// TwinCAT 3 PLC project Controller
// ProgramVersion: 3.1.4026.15
// libraries:
//   Tc2_Math, * (Beckhoff Automation GmbH)
//   Tc2_MC2, * (Beckhoff Automation GmbH)
//   Tc2_MC2_Camming, * (Beckhoff Automation GmbH)
//   Tc2_Standard, * (Beckhoff Automation GmbH)
//   Tc2_System, * (Beckhoff Automation GmbH)
//   Tc2_Utilities, * (Beckhoff Automation GmbH)
//   Tc3_Module, * (Beckhoff Automation GmbH)
// project tree:
//   DUTs/ ST_RECIPE_VARIABLES.TcDUT, ST_WORKER_VARIABLES.TcDUT
//   GVLs/ GVL.TcGVL
//   / PlcTask.TcTTO
//   POUs/ FB_CamProfiles.TcPOU, FB_MasterCamControl.TcPOU, MAIN.TcPOU
// real-time tasks:
//   TASK PlcTask: cycle T#10ms, priority 20, ADS port 350
// motion (NC):
//   TASK NC-Task 1 SAF: cycle T#2ms, priority 4, ADS port 501
//   TASK NC-Task 1 SVB: cycle T#10ms, priority 8, ADS port 511
//   AXIS Master (id 1)
//     Velo: Maximum=10000
//     OtherSettings: AllowMotionCmdToSlave=true
//     encoder EncType=1
//     drive DrvType=5
//       Analog: TorqueSetpointScale=10, ScaleFactorActTorque=0.1
//       TimeComp: TaskDelayCycles=1
//     controller CtrType=1
//       CtrPara: PriorControlFactor=1
//         Observer: BandWidth=20
//   AXIS Slave_1 (id 2)
//     OtherSettings: AllowMotionCmdToSlave=true
//     encoder EncType=1
//     drive DrvType=5
//       Analog: TorqueSetpointScale=10, ScaleFactorActTorque=0.1
//       TimeComp: TaskDelayCycles=1
//     controller CtrType=1
//       CtrPara: PriorControlFactor=1
//         Observer: BandWidth=20
//   AXIS Slave_2 (id 3)
//     OtherSettings: AllowMotionCmdToSlave=true
//     encoder EncType=1
//     drive DrvType=5
//       Analog: TorqueSetpointScale=10, ScaleFactorActTorque=0.1
//       TimeComp: TaskDelayCycles=1
//     controller CtrType=1
//       CtrPara: PriorControlFactor=1
//         Observer: BandWidth=20
//   AXIS Slave_3 (id 4)
//     OtherSettings: AllowMotionCmdToSlave=true
//     encoder EncType=1
//     drive DrvType=5
//       Analog: TorqueSetpointScale=10, ScaleFactorActTorque=0.1
//       TimeComp: TaskDelayCycles=1
//     controller CtrType=1
//       CtrPara: PriorControlFactor=1
//         Observer: BandWidth=20
//   AXIS Slave_4 (id 5)
//     OtherSettings: AllowMotionCmdToSlave=true
//     encoder EncType=1
//     drive DrvType=5
//       Analog: TorqueSetpointScale=10, ScaleFactorActTorque=0.1
//       TimeComp: TaskDelayCycles=1
//     controller CtrType=1
//       CtrPara: PriorControlFactor=1
//         Observer: BandWidth=20
// variable links:
//   Controller/Controller Instance <-> NC-Task 1 SAF/Axes/Master
//     PlcTask Inputs/GVL.Master.NcToPlc <-> Outputs/ToPlc
//     PlcTask Outputs/GVL.Master.PlcToNc <-> Inputs/FromPlc
//   Controller/Controller Instance <-> NC-Task 1 SAF/Axes/Slave_1
//     PlcTask Inputs/GVL.Slave_1.NcToPlc <-> Outputs/ToPlc
//     PlcTask Outputs/GVL.Slave_1.PlcToNc <-> Inputs/FromPlc
//   Controller/Controller Instance <-> NC-Task 1 SAF/Axes/Slave_2
//     PlcTask Inputs/GVL.Slave_2.NcToPlc <-> Outputs/ToPlc
//     PlcTask Outputs/GVL.Slave_2.PlcToNc <-> Inputs/FromPlc
//   Controller/Controller Instance <-> NC-Task 1 SAF/Axes/Slave_3
//     PlcTask Inputs/GVL.Slave_3.NcToPlc <-> Outputs/ToPlc
//     PlcTask Outputs/GVL.Slave_3.PlcToNc <-> Inputs/FromPlc
//   Controller/Controller Instance <-> NC-Task 1 SAF/Axes/Slave_4
//     PlcTask Inputs/GVL.Slave_4.NcToPlc <-> Outputs/ToPlc
//     PlcTask Outputs/GVL.Slave_4.PlcToNc <-> Inputs/FromPlc

CONFIGURATION Controller
    RESOURCE PLC ON TwinCAT3
        TASK PlcTask(INTERVAL := T#10ms, PRIORITY := 20);
        PROGRAM MAIN WITH PlcTask : MAIN;
    END_RESOURCE
END_CONFIGURATION

// ---- DUTs/ST_RECIPE_VARIABLES.TcDUT
TYPE ST_RECIPE_VARIABLES :
STRUCT
	sRecipeName			: STRING;
	MotionPoints_CAM_1	: ARRAY [0..360, 0..1] OF REAL;
	MotionPoints_CAM_2	: ARRAY [0..360, 0..1] OF REAL;
	MotionPoints_CAM_3	: ARRAY [0..360, 0..1] OF REAL;
	MotionPoints_CAM_4	: ARRAY [0..360, 0..1] OF REAL;
	// And other Recipe Variables
	bCheckBool			: BOOL;
	nTestInt			: INT;
	rTestReal			: REAL;
	lrTestLReal			: LREAL;
	udnAnotherInt		: UDINT;
END_STRUCT
END_TYPE

// ---- DUTs/ST_WORKER_VARIABLES.TcDUT
TYPE ST_WORKER_VARIABLES :
STRUCT
	sMachineName		: STRING := 'Worker_1';
	sProgramVersion		: STRING := '1.0';
	stRecipeVariables	: ST_RECIPE_VARIABLES;
	
	eStatus				: (IDLE,
							ASSIGNED,
							RUNNING,
							MAINTAINANCE_REQ);
	
	bGetRecipeAndCams	: BOOL;
	bCamsReady			: BOOL;
	sAssignedRecipe		: STRING;
	udnNumberOfJobsDone	: UDINT;
	udnDaysSinceServiced: UDINT;
END_STRUCT
END_TYPE

// ---- GVLs/GVL.TcGVL
{attribute 'qualified_only'}
VAR_GLOBAL
	Master		: AXIS_REF;		// Master will be a virtual axis
	rMasterVel	: REAL;
	
	// The 4 slaves will be the 4 Beckhoff motors
	Slave_1		: AXIS_REF;
	Slave_2		: AXIS_REF;
	Slave_3		: AXIS_REF;
	Slave_4		: AXIS_REF;
END_VAR

// ---- POUs/MAIN.TcPOU
PROGRAM MAIN
VAR
	stWorker_1		: ST_WORKER_VARIABLES;
	stRecipe		: ST_RECIPE_VARIABLES;
	
	// Slave positions for the cam table
	// Array [1..4] are slaves 1 - 4, each of the slave is a 2d array **REQUIRED by cam table ref**
	// Array [0..359] are master-slave position pair
	ALL_CAM			: ARRAY [1..4] OF ARRAY [0..359] OF ARRAY [0..1] OF LREAL;		
	ALL_CAM_REF		: ARRAY [1..4] OF MC_CAM_REF;		// Cam table reference
	
	nState			: INT;
	bStart			: BOOL;
	
	fbMasterCam		: FB_MasterCamControl;
	fbCamProfiles	: FB_CamProfiles;
	mcHome			: MC_Home;
	bMasterRun		: BOOL;
	bHalt			: BOOL;
	bReset			: BOOL;
	bReadDone		: BOOL;
	bCreateDone		: BOOL;
	
	bCamIn			: BOOL;
	nUpdate			: INT;
END_VAR

fbMasterCam();

CASE nState OF
	0:	// IDLE
		IF bStart THEN
			nState		:= 5;
		END_IF
	5:	// Initialize and enable the power on Master and Slaves Axes
		fbMasterCam.mInitialize(TRUE);
		IF fbMasterCam.pInitialized THEN
			fbMasterCam.mInitialize(FALSE);
			nState		:= 10;
		END_IF
	(**************** These will not be implemented in the real project ***********)
	(**************** recipe management will replace the csv file *****************)
	10:	// Read CAM profiles from CSV files and store in CAM arrays
		fbCamProfiles.mReadAndStoreSlavePositions(TRUE, ALL_CAM);
		IF fbCamProfiles.pReadDone THEN
			fbCamProfiles.mReadAndStoreSlavePositions(FALSE, ALL_CAM);
			nState		:= 15;
		END_IF
	15:	// Create Twincat digital CAM tables from CAM profile arrays
		fbCamProfiles.mCreateCamProfiles(TRUE, ALL_CAM, ALL_CAM_REF);
		IF fbCamProfiles.pCreateDone THEN
			fbCamProfiles.mCreateCamProfiles(FALSE, ALL_CAM, ALL_CAM_REF);
			GVL.rMasterVel:= 0.5;			// Start Master at minimum speed
			bMasterRun	:= TRUE;			// to couple CAM profiles
			fbMasterCam.pRunCams:= TRUE;	// Start Slaves
			nState		:= 20;
		END_IF
	(**************      ~30s to complete the csv reading     *********************)
	(******************************************************************************)
	20:	// Assign CAM tables to their respective Slave Axes
		fbMasterCam.mMultiCamIn(TRUE);
		IF fbMasterCam.pCamInDone THEN
			fbMasterCam.mMultiCamIn(TRUE);
			nState		:= 25;
		END_IF
	25:	// Speed up Master after all CAMs done coupling 
		IF NOT bMasterRun THEN
			GVL.rMasterVel	:= 180;
			bMasterRun		:= TRUE;
			nState			:= 26;
		END_IF
		
	(********************* Not used *******************)
	30:	// Stop all axes
		fbMasterCam.mHalt(bHalt);
	35: // Reset all axes
		fbMasterCam.mReset(bReset);
END_CASE
fbMasterCam.mRun(bMasterRun);

METHOD mLoadCSVToCAMs : BOOL
//VAR_INPUT
//	Execute		: BOOL;
//END_VAR
//VAR_IN_OUT
//	Slave_CAM	: ARRAY [0..360] OF ARRAY [0..1] OF LREAL;
//END_VAR
//CASE nState OF
//	0:
//		IF Execute THEN
//			sReadLine	:= '';
//			nStringIndex:= 0;
//			nState		:= 1;
//		END_IF
//	1:
//		fbFileOpen(
//			sNetId		:= '10.75.0.183.1.1',
//			sPathName	:= sFilePath,
//			nMode		:= FOPEN_MODEREAD,
//			ePath		:= PATH_GENERIC,
//			bExecute	:= TRUE,
//			tTimeout	:= DEFAULT_ADS_TIMEOUT);
//		nState			:= 2;
//	2:
//		fbFileOpen(	
//			bExecute 	:= FALSE,
//			hFile 		=> fileHandle);
//		IF NOT fbFileOpen.bBusy THEN
//			IF NOT fbFileOpen.bError THEN
//				nState	:= 5;
//			ELSE
//				nState	:= 255;
//			END_IF
//		END_IF
//	5:
//		fbFileGets(
//			sNetId		:= '10.75.0.183.1.1',
//			hFile		:= fileHandle,
//			bExecute	:= TRUE,
//			sLine		=> sReadLine);
//		IF NOT fbFileGets.bBusy AND NOT fbFileGets.bError THEN
//			fbFileGets(bExecute:=FALSE);
//			IF NOT fbFileGets.bEOF THEN
//				nState	:= 10;
//			ELSE
//				nStringIndex:= 0;
//				nState	:= 15;
//			END_IF
//		ELSIF fbFileGets.bError THEN
//				nState	:= 255;
//		END_IF
//	10:
//		arrString[nStringIndex]:= sReadLine;
//		nStringIndex	:= nStringIndex + 1;
//		nState			:= 5;
//	15:
//		FOR nStringIndex := 0 TO 360 DO
//			rAbsPosition:= STRING_TO_REAL(arrString[nStringIndex]);
//			arrTemp[0]	:= nStringIndex;
//			arrTemp[1]	:= rAbsPosition;
//			Slave_CAM[nStringIndex]:= arrTemp;
//		END_FOR
//		nState			:= 60;
		
//	60:
//		fbFileClose(
//			sNetId		:= '10.75.0.183.1.1',
//			hFile		:= fileHandle,
//			bExecute	:= TRUE);
//		nState			:= 61;
//	61:
//		fbFileClose(bExecute:=FALSE);
//		IF NOT fbFileClose.bBusy THEN
//			IF NOT fbFileClose.bError THEN
//				nState	:= 62;
//			ELSE
//				nState	:= 255;
//			END_IF
//		END_IF
//	62:
//		sTemp			:= '';
//		sFilePath		:= 'C:\';
//		bExecute		:= FALSE;
//		nState			:= 0;
//END_CASE
END_METHOD

END_PROGRAM

// ---- POUs/FB_MasterCamControl.TcPOU
FUNCTION_BLOCK FB_MasterCamControl
VAR_INPUT
END_VAR
VAR_OUTPUT
END_VAR
VAR
//	fbMaster		: CAM_AXIS_BASE;
//	fbSlave_1		: CAM_AXIS_BASE;
//	fbSlave_2		: CAM_AXIS_BASE;
//	fbSlave_3		: CAM_AXIS_BASE;
//	fbSlave_4		: CAM_AXIS_BASE;
	mcHome			: MC_Home;
	bRunCams		: BOOL;
	
	bInitialized	: BOOL;
	bCamInDone		: BOOL;
END_VAR

//fbMaster.mRunCam(bRunCams);
//fbSlave_1.mRunCam(bRunCams);
//fbSlave_2.mRunCam(bRunCams);
//fbSlave_3.mRunCam(bRunCams);
//fbSlave_4.mRunCam(bRunCams);

// Reset Virtual Master Cam to 0 after 1 complete revolution
IF GVL.Master.NcToPlc.ModuloSetTurns = 1 AND NOT mcHome.Done THEN
	mcHome(
		Axis		:= GVL.Master,
		Execute		:= TRUE,
		Position	:= 0,
		HomingMode	:= MC_Direct);
ELSIF mcHome.Done THEN
	mcHome(Axis := GVL.Master, Execute := FALSE);
END_IF

METHOD mCamOut : BOOL
VAR_INPUT
	Execute		: BOOL;
END_VAR

VAR_INST
	CamOut		: MC_CamOut;
	
	nState		: INT;
	rtStart		: R_TRIG;
END_VAR
CASE nState OF
	0:
		rtStart(CLK := Execute);
		IF rtStart.Q THEN
			mCamOut		:= FALSE;
			nState		:= 5;
		END_IF
	5:
		CamOut(Slave := GVL.Slave_1, Execute := TRUE);
		IF CamOut.Done THEN
			CamOut(Slave := GVL.Slave_1, Execute := FALSE);
			nState		:= 15;
		END_IF
	15:
		CamOut(Slave := GVL.Slave_2, Execute := TRUE);
		IF CamOut.Done THEN
			CamOut(Slave := GVL.Slave_2, Execute := FALSE);
			nState		:= 20;
		END_IF
	20:
		CamOut(Slave := GVL.Slave_3, Execute := TRUE);
		IF CamOut.Done THEN
			CamOut(Slave := GVL.Slave_3, Execute := FALSE);
			nState		:= 25;
		END_IF
	25:
		CamOut(Slave := GVL.Slave_4, Execute := TRUE);
		IF CamOut.Done THEN
			CamOut(Slave := GVL.Slave_4, Execute := FALSE);
			nState		:= 30;
		END_IF
	30:
		mCamOut			:= TRUE;
		nState			:= 0;
END_CASE
END_METHOD

METHOD mHalt : BOOL
VAR_IN_OUT
	Execute		: BOOL;
END_VAR
VAR_INST
	HaltMaster	: MC_Halt;
	HaltSlave_1	: MC_Halt;
	HaltSlave_2	: MC_Halt;
	HaltSlave_3	: MC_Halt;
	HaltSlave_4	: MC_Halt;
END_VAR
HaltMaster(Axis := GVL.Master, Execute := Execute);
HaltSlave_1(Axis := GVL.Slave_1, Execute := Execute);
HaltSlave_2(Axis := GVL.Slave_2, Execute := Execute);
HaltSlave_3(Axis := GVL.Slave_3, Execute := Execute);
HaltSlave_4(Axis := GVL.Slave_4, Execute := Execute);

IF HaltMaster.Done AND HaltSlave_1.Done AND HaltSlave_2.Done AND HaltSlave_3.Done AND HaltSlave_4.Done THEN
	Execute := FALSE;
END_IF
END_METHOD

(* Move all axes to 0 position *)
METHOD mHomeAxes : BOOL
VAR_INPUT
	Execute			: BOOL;
END_VAR

VAR_INST
	MoveHome		: MC_MoveAbsolute;
	mcHome			: MC_Home;
	
	nState			: INT;
	rtStart			: R_TRIG;
END_VAR
CASE nState OF
	0:
		rtStart(CLK := Execute);
		IF rtStart.Q THEN
			mHomeAxes	:= FALSE;
			nState		:= 5;
		END_IF
	5:
		MoveHome(
			Axis		:= GVL.Slave_1,
			Execute		:= TRUE,
			Position	:= 0,
			Velocity	:= 2000);
		IF MoveHome.Done THEN
			MoveHome(Axis := GVL.Slave_1, Execute := FALSE);
			nState		:= 10;
		END_IF
	10:
		MoveHome(
			Axis		:= GVL.Slave_2,
			Execute		:= TRUE,
			Position	:= 0,
			Velocity	:= 2000);
		IF MoveHome.Done THEN
			MoveHome(Axis := GVL.Slave_2, Execute := FALSE);
			nState		:= 15;
		END_IF
	15:
		MoveHome(
			Axis		:= GVL.Slave_3,
			Execute		:= TRUE,
			Position	:= 0,
			Velocity	:= 2000);
		IF MoveHome.Done THEN
			MoveHome(Axis := GVL.Slave_3, Execute := FALSE);
			nState		:= 20;
		END_IF
	20:
		MoveHome(
			Axis		:= GVL.Slave_4,
			Execute		:= TRUE,
			Position	:= 0,
			Velocity	:= 2000);
		IF MoveHome.Done THEN
			MoveHome(Axis := GVL.Slave_4, Execute := FALSE);
			nState		:= 25;
		END_IF
	25:
		mcHome(
			Axis		:= GVL.Master,
			Execute		:= TRUE,
			Position	:= 0,
			HomingMode	:= MC_Direct);
		IF mcHome.Done THEN
			mcHome(Axis := GVL.Master, Execute := FALSE);
			nState		:= 30;
		END_IF
	30:
		mHomeAxes		:= TRUE;
		nState			:= 0;
END_CASE
END_METHOD

METHOD mInitialize : BOOL
VAR_INPUT
	Execute			: BOOL;
END_VAR
VAR_INST
	nState			: INT;
	rtStart			: R_TRIG;
END_VAR
CASE nState OF
	0:
		rtStart(CLK := Execute);
		IF rtStart.Q THEN
			bInitialized	:= FALSE;
			nState			:= 1;
		END_IF
	1:
		IF mCamOut(TRUE) THEN
			mCamOut(FALSE);
			nState			:= 5;
		END_IF
	5:
		IF mReset(TRUE) THEN
			mReset(FALSE);
			nState			:= 10;
		END_IF
	10:
		IF mPower(TRUE) THEN
			mPower(FALSE);
			nState			:= 15;
		END_IF
	15:
		IF mHomeAxes(TRUE) THEN
			mHomeAxes(FALSE);
			nState			:= 100;
		END_IF
	100:
		bInitialized		:= TRUE;
		nState				:= 0;
END_CASE
END_METHOD

METHOD mMultiCamIn : BOOL
VAR_INPUT
	Execute		: BOOL;
END_VAR

VAR_INST
	nState		: INT;
	rtStart		: R_TRIG;
	
	CamIn		: MC_CamIn;
	
	Options		: ST_CamInOptions;
END_VAR
CASE nState OF
	0:
		rtStart(CLK := Execute);
		IF rtStart.Q THEN
			Options.ActivationMode:= MC_CAMACTIVATION_INSTANTANEOUS;
			Options.InterpolationType:= MC_INTERPOLATIONTYPE_LINEAR;
			bCamInDone	:= FALSE;
			nState		:= 5;
		END_IF
	5:
		CamIn(
			Master		:= GVL.Master,
			Slave		:= GVL.Slave_1,
			Execute		:= TRUE,
 			StartMode	:= MC_STARTMODE_ABSOLUTE,
			Options		:= Options,
			CamTableID	:= 1);
		IF CamIn.InSync THEN
			CamIN(Master:= GVL.Master, Slave:= GVL.Slave_1, Execute:= FALSE);
			nState		:= 10;
		END_IF
	10:
		CamIn(
			Master		:= GVL.Master,
			Slave		:= GVL.Slave_2,
			Execute		:= TRUE,
			StartMode	:= MC_STARTMODE_ABSOLUTE,
			Options		:= Options,
			CamTableID	:= 2);
		IF CamIn.InSync THEN
			CamIN(Master:= GVL.Master, Slave:= GVL.Slave_2, Execute:= FALSE);
			nState		:= 15;
		END_IF
	15:
		CamIn(
			Master		:= GVL.Master,
			Slave		:= GVL.Slave_3,
			Execute		:= TRUE,
			StartMode	:= MC_STARTMODE_ABSOLUTE,
			Options		:= Options,
			CamTableID	:= 3);
		IF CamIn.InSync THEN
			CamIN(Master:= GVL.Master, Slave:= GVL.Slave_3, Execute:= FALSE);
			nState		:= 20;
		END_IF
	20:
		CamIn(
			Master		:= GVL.Master,
			Slave		:= GVL.Slave_4,
			Execute		:= TRUE,
			StartMode	:= MC_STARTMODE_ABSOLUTE,
			Options		:= Options,
			CamTableID	:= 4);
		IF CamIn.InSync THEN
			CamIN(Master:= GVL.Master, Slave:= GVL.Slave_4, Execute:= FALSE);
			nState		:= 25;
		END_IF
	25:
		bCamInDone		:= TRUE;
		nState			:= 0;
END_CASE
END_METHOD

METHOD mPower : BOOL
VAR_INPUT
	Execute			: BOOL;
END_VAR
VAR_INST
	nState			: INT;
	rtStart			: R_TRIG;
	
	PowerMaster				: MC_Power;
	PowerSlave_1			: MC_Power;
	PowerSlave_2			: MC_Power;
	PowerSlave_3			: MC_Power;
	PowerSlave_4			: MC_Power;
END_VAR
CASE nState OF
	0:
		rtStart(CLK := Execute);
		IF rtStart.Q THEN
			mPower			:= FALSE;
			nState			:= 5;
		END_IF
	5:
		PowerMaster(
			Axis			:= GVL.Master,
			Enable			:= TRUE,
			Enable_Positive	:= TRUE,
			Enable_Negative	:= TRUE);
		IF PowerMaster.Status THEN			// Status = Done (BOOL)
			nState			:= 10;
		END_IF
	10:
		PowerSlave_1(
			Axis			:= GVL.Slave_1,
			Enable			:= TRUE,
			Enable_Positive	:= TRUE,
			Enable_Negative	:= TRUE);
		IF PowerSlave_1.Status THEN
			nState			:= 15;
		END_IF
	15:
		PowerSlave_2(
			Axis			:= GVL.Slave_2,
			Enable			:= TRUE,
			Enable_Positive	:= TRUE,
			Enable_Negative	:= TRUE);
		IF PowerSlave_2.Status THEN
			nState			:= 20;
		END_IF
	20:
		PowerSlave_3(
			Axis			:= GVL.Slave_3,
			Enable			:= TRUE,
			Enable_Positive	:= TRUE,
			Enable_Negative	:= TRUE);
		IF PowerSlave_3.Status THEN
			nState			:= 25;
		END_IF
	25:
		PowerSlave_4(
			Axis			:= GVL.Slave_4,
			Enable			:= TRUE,
			Enable_Positive	:= TRUE,
			Enable_Negative	:= TRUE);
		IF PowerSlave_4.Status THEN
			nState			:= 100;
		END_IF
	100:
		mPower				:= TRUE;
		nState				:= 0;
END_CASE
END_METHOD

METHOD mReset : BOOL
VAR_INPUT
	Execute		: BOOL;
END_VAR
VAR_INST
//	ResetMaster	: MC_Reset;
//	ResetSlave_1: MC_Reset;
//	ResetSlave_2: MC_Reset;
//	ResetSlave_3: MC_Reset;
//	ResetSlave_4: MC_Reset;
	Reset		: MC_Reset;	

	nState		: INT;
	rtStart		: R_TRIG;
END_VAR
CASE nState OF
	0:
		rtStart(CLK := Execute);
		IF rtStart.Q THEN
			mReset	:= FALSE;
			nState	:= 10;
		END_IF
	10:
		Reset(Axis := GVL.Master, Execute := Execute);
		IF Reset.Done THEN
			Reset(Axis := GVL.Master, Execute := FALSE);
			nState	:= 15;
		END_IF
	15:
		Reset(Axis := GVL.Slave_1, Execute := Execute);
		IF Reset.Done THEN
			Reset(Axis := GVL.Slave_1, Execute := FALSE);
			nState	:= 20;
		END_IF
	20:
		Reset(Axis := GVL.Slave_2, Execute := Execute);
		IF Reset.Done THEN
			Reset(Axis := GVL.Slave_2, Execute := FALSE);
			nState	:= 25;
		END_IF
	25:
		Reset(Axis := GVL.Slave_3, Execute := Execute);
		IF Reset.Done THEN
			Reset(Axis := GVL.Slave_3, Execute := FALSE);
			nState	:= 30;
		END_IF
	30:
		Reset(Axis := GVL.Slave_4, Execute := Execute);
		IF Reset.Done THEN
			Reset(Axis := GVL.Slave_4, Execute := FALSE);
			nState	:= 35;
		END_IF
	35:
		mReset		:= TRUE;
		nState		:= 0;
END_CASE


//ResetMaster(Axis := Master, Execute := Execute);
//ResetSlave_1(Axis := Slave_1, Execute := Execute);
//ResetSlave_2(Axis := Slave_2, Execute := Execute);
//ResetSlave_3(Axis := Slave_3, Execute := Execute);
//ResetSlave_4(Axis := Slave_4, Execute := Execute);

//IF ResetMaster.Done AND ResetSlave_1.Done AND ResetSlave_2.Done AND ResetSlave_3.Done AND ResetSlave_4.Done THEN
//	Execute	:= FALSE;
//END_IF
END_METHOD

METHOD mRun : BOOL
VAR_INPUT
END_VAR
VAR_IN_OUT
	bMasterRun		: BOOL;
END_VAR
VAR_INST
	nState			: INT;
	rtRerun			: R_TRIG;
	
	MoveMaster 		: MC_MoveVelocity;
	
	MoveSlave_1		: MC_MoveAbsolute;
	MoveSlave_2		: MC_MoveAbsolute;
	MoveSlave_3		: MC_MoveAbsolute;
	MoveSlave_4		: MC_MoveAbsolute;
END_VAR
IF bMasterRun THEN
	MoveMaster(
		Axis		:= GVL.Master,
		Execute		:= TRUE,
		Velocity	:= GVL.rMasterVel,
		Direction	:= MC_Positive_Direction);
	IF MoveMaster.InVelocity THEN
		MoveMaster(Axis := GVL.Master, Execute := FALSE);
		bMasterRun	:= FALSE;
	END_IF
END_IF

MoveSlave_1(
	Axis		:= GVL.Slave_1,
	Execute		:= bRunCams,
	Position	:= 0,
	Velocity	:= 1000);
MoveSlave_2(
	Axis		:= GVL.Slave_2,
	Execute		:= bRunCams,
	Position	:= 0,
	Velocity	:= 1000);
MoveSlave_3(
	Axis		:= GVL.Slave_3,
	Execute		:= bRunCams,
	Position	:= 0,
	Velocity	:= 1000);
MoveSlave_4(
	Axis		:= GVL.Slave_4,
	Execute		:= bRunCams,
	Position	:= 0,
	Velocity	:= 1000);
END_METHOD

PROPERTY pCamInDone : BOOL
GET
pCamInDone := bCamInDone;
END_GET
END_PROPERTY

PROPERTY pInitialized : BOOL
GET
pInitialized := bInitialized;
END_GET
END_PROPERTY

PROPERTY pRunCams : BOOL
GET
pRunCams := bRunCams;
END_GET
SET
bRunCams := pRunCams;
END_SET
END_PROPERTY

END_FUNCTION_BLOCK

// ---- POUs/FB_CamProfiles.TcPOU
(* This whole function block is to load cam profiles from a csv file
 * onto the PLC program. This is only temporarily needed to test/learn the cam library.
 * This will not be used when developing the machine, since the cam profiles will be loaded
 * from recipe management.
 *)

FUNCTION_BLOCK FB_CamProfiles
VAR_INPUT
END_VAR
VAR_OUTPUT
END_VAR
VAR
	sFilePath		: STRING;
	
	bReadDone		: BOOL;
	bCreateDone		: BOOL;
END_VAR

METHOD mCreateCamProfiles : BOOL
VAR_INPUT
	Execute			: BOOL;
END_VAR
VAR_IN_OUT
	ALL_CAM			: ARRAY [1..4] OF ARRAY [0..359] OF ARRAY [0..1] OF LREAL;
	ALL_CAM_REF		: ARRAY [1..4] OF MC_CAM_REF;
END_VAR

VAR_INST
	nState			: INT;
	rtStart			: R_TRIG;
	
	nIndex			: INT;
	CamTableSelect	: MC_CamTableSelect;
END_VAR
CASE nState OF
	0:
		rtStart(CLK := Execute);
		IF rtStart.Q THEN
			bCreateDone	:= FALSE;
			nState		:= 5;
		END_IF
	5:
		FOR nIndex := 1 TO 4 DO
			ALL_CAM_REF[nIndex].pArray		:= ADR(ALL_CAM[nIndex]);
			ALL_CAM_REF[nIndex].ArraySize	:= SIZEOF(ALL_CAM[nIndex]);
			ALL_CAM_REF[nIndex].TableType	:= MC_TABLETYPE_EQUIDISTANT;
			ALL_CAM_REF[nIndex].NoOfRows	:= 360;
			ALL_CAM_REF[nIndex].NoOfColumns	:= 2;
		END_FOR
		nIndex 			:= 1;
		nState			:= 10;
	10:
		CamTableSelect(
			Execute		:= TRUE,
			Periodic	:= FALSE,
			CamTableID	:= nIndex,
			CamTable	:= ALL_CAM_REF[nIndex]);
		IF CamTableSelect.Error THEN 
			nState		:= 255;
		ELSIF CamTableSelect.Done AND nIndex < 4 THEN
			CamTableSelect(Execute:=FALSE, CamTable	:= ALL_CAM_REF[nIndex]);
			nIndex		:= nIndex + 1;
		ELSIF CamTableSelect.Done THEN
			CamTableSelect(Execute:=FALSE, CamTable	:= ALL_CAM_REF[nIndex]);
			nState		:= 15;
		END_IF
	15:
		bCreateDone		:= TRUE;
		nState			:= 0;
END_CASE
END_METHOD

METHOD mReadAndStoreSlavePositions : BOOL
VAR_INPUT
	Execute			: BOOL;
END_VAR

VAR_IN_OUT
	ALL_CAM			: ARRAY [1..4] OF ARRAY [0..359] OF ARRAY [0..1] OF LREAL;
END_VAR

VAR_INST
	nState			: INT;
	rtStart			: R_TRIG;
	fbFileOpen		: FB_FileOpen;
	fbFileClose		: FB_FileClose;
	fbFileGets		: FB_FileGets;	// Read 1 csv line function block.
	fileHandle		: UINT;
	
	sReadLine		: STRING;
	
	aPositionStr	: ARRAY [0..360] OF STRING;
	nIndex			: INT;
	nCamFileNumber	: INT := 1;
	lrAbsPosition	: LREAL;
	aTemp			: ARRAY [0..1] OF LREAL;
END_VAR
CASE nState OF
	0:	// IDLE
		rtStart(CLK := Execute);
		IF rtStart.Q THEN
			bReadDone	:= FALSE;
			sReadLine	:= '';
			nIndex		:= 0;
			nState		:= 5;
		END_IF
	5:	// Set file path base Cam profile
		sFilePath		:= 'C:\Users\Administrator\Desktop\Cam_Profiles\8605-005 V2\Slave_';// Path: 	.\
		sFilePath		:= CONCAT(sFilePath, INT_TO_STRING(nCamFileNumber));				//			.\Slave_#
		sFilePath		:= CONCAT(sFilePath, '.csv');										//			.\Slave_#.csv
		nState			:= 10;
	10:	// Open the correspondence CSV file
		fbFileOpen(
			sNetId		:= '10.75.0.183.1.1',
			sPathName	:= sFilePath,
			nMode		:= FOPEN_MODEREAD,
			ePath		:= PATH_GENERIC,
			bExecute	:= TRUE,
			tTimeout	:= DEFAULT_ADS_TIMEOUT);
		nState			:= 15;
	15:	// File open helper state
		fbFileOpen(	bExecute := FALSE, hFile => fileHandle);
		IF NOT fbFileOpen.bBusy AND NOT fbFileOpen.bError THEN
			nState		:= 20;
		ELSIF fbFileOpen.bError THEN
			nState		:= 255;
		END_IF
	20:	// Read 1 line from the openned file, store the line to sReadLine
		fbFileGets(
			sNetId		:= '10.75.0.183.1.1',
			hFile		:= fileHandle,
			bExecute	:= TRUE,
			sLine		=> sReadLine);
		IF NOT fbFileGets.bBusy AND NOT fbFileGets.bError THEN
			// Reset fbFileGets execute flag => remove the read line from memory buffer, so when fbFileGets is called again, the next line is read.
			fbFileGets(bExecute:=FALSE);
			// If not End_Of_File, then append the value to the Position Array and increment the index.
			IF NOT fbFileGets.bEOF THEN
				aPositionStr[nIndex]:= sReadLine;
				nIndex	:= nIndex + 1;
			ELSE
				nIndex	:= 0;
				nState	:= 25;
			END_IF
		ELSIF fbFileGets.bError THEN
				nState	:= 255;
		END_IF
	25:	// 
		FOR nIndex := 0 TO 359 DO
			lrAbsPosition:= STRING_TO_LREAL(aPositionStr[nIndex]);
			aTemp[0]	:= nIndex;
			aTemp[1]	:= lrAbsPosition;
			ALL_CAM[nCamFileNumber][nIndex]:= aTemp;
		END_FOR
		nState			:= 30;
	30:
		nIndex 			:= 0;
		fbFileClose(
			sNetId		:= '10.75.0.183.1.1',
			hFile		:= fileHandle,
			bExecute	:= TRUE);
		nState			:= 35;
	35:
		fbFileClose(bExecute:=FALSE);
		IF NOT fbFileClose.bBusy THEN
			IF NOT fbFileClose.bError THEN
				nState	:= 40;
			ELSE
				nState	:= 255;
			END_IF
		END_IF
	40:
		IF nCamFileNumber < 4 THEN
			nCamFileNumber:= nCamFileNumber + 1;
			nState		:= 5;
		ELSE
			bReadDone	:= TRUE;
			nState		:= 0;
		END_IF
END_CASE
END_METHOD

PROPERTY pCreateDone : BOOL
GET
pCreateDone := bCreateDone;
END_GET
END_PROPERTY

PROPERTY pReadDone : BOOL
GET
pReadDone := bReadDone;
END_GET
END_PROPERTY

END_FUNCTION_BLOCK
